FUNCTION TryConvert_LINT_TO_LWORD : BOOL
VAR_INPUT
	in : LINT;
	out : REFERENCE TO LWORD;
END_VAR

IF in < DatatypeLimits.MIN_VALUE_OF_LINT_WHICH_CAN_BE_HELD_IN_A_LWORD THEN
	RETURN;
END_IF

out := LINT_TO_LWORD(in);
TryConvert_LINT_TO_LWORD := TRUE;

END_FUNCTION

(* stored: Version 1.1.0.1, ProductVersion 3.1.4024.12
   POU TryConvert_LINT_TO_LWORD: Id {89503f33-0d4f-4293-a700-e09eeba3535e}, SpecialFunc None *)
